VAR_GLOBAL
	// Axes
    M1: DUT_MotionStage:=(nCommand:=3); // Yup
	M2: DUT_MotionStage:=(nCommand:=3); // Ydwn
	M3: DUT_MotionStage:=(nCommand:=3); // Xup
	M4: DUT_MotionStage:=(nCommand:=3); // Xdwn
	M5: DUT_MotionStage:=(nCommand:=3); // PitchCoarse
	M1_Extras : DUT_MotionStage_Extras;
	M2_Extras : DUT_MotionStage_Extras;
	M3_Extras : DUT_MotionStage_Extras;
	M4_Extras : DUT_MotionStage_Extras;
	M5_Extras : DUT_MotionStage_Extras;

	M1L0_Pitch	    :	HOMS_PitchMechanism := (
		ReqPosLimHi := 56000,
		ReqPosLimLo := 54150,
		diEncPosLimHi := 10126850,
		diEncPosLimLo := 9727550);
END_VAR

(* stored: Version 1.1.0.1, ProductVersion 3.1.4022.18
   GVL GVL_Devices: Id {cb7cf638-cc80-4f58-a532-470704faedf8} *)
